# EPICS substitutions: template/mch_type1_ess.substitutions
#
# Type 1 : MCH
#          This is the standard ESS MCH for 9U/3U MTCA crate
#
#
# MCH (0)
# Manufacturer(12)         : Schroff GmbH
# Board Name(37)           : Schroff MicroTCA Backplane horizontal
# Manufacturer(12)         : Schroff GmbH
# Product Name(22)         : Schroff MicroTCA Shelf
# NAT-MCH (3)
# Manufacturer(21)         : N.A.T. GmbH - Germany
# Board Name(07)           : NAT-MCH
# Clock (60)
# Manufacturer(21)         : N.A.T. GmbH - Germany
# Product Name(16)         : NAT-MCH-CLK-PHYS
# HubMod1 (61)
# Manufacturer(21)         : N.A.T. GmbH - Germany
# Product Name(15)         : PCIe Hub Module

# show_fru
#  0   MCH       M4    NMCH-CM
#  3   mcmc1     M4    NAT-MCH-MCMC
# 60   Clock1    M4    MCH-Clock
# 61   HubMod1   M4    MCH-PCIe

# nat> show_sensorinfo 0
# Sensor Information for NMCH-CM
# ==================================================================
#   #   SDRType  Sensor Entity Inst  Value   State    Name
# ------------------------------------------------------------------
#   -   MDevLoc          0xc2  0x66                    NMCH-CM
#   0   Compact  0xf0    0xc2  0x66  0x10              HS 000 CM
# ------------------------------------------------------------------
# nat> show_sensorinfo 3
# Sensor Information for FRU 3 / MCMC1
# ==================================================================
#   #   SDRType  Sensor Entity Inst  Value   State    Name
# ------------------------------------------------------------------
#   -   MDevLoc          0xc2  0x61                    NAT-MCH-MCMC
#   1   Full     Temp    0xc2  0x61  36 C       ok     Temp CPU
#   2   Full     Temp    0xc2  0x61  32 C       ok     Temp I/O
#   3   Compact  0xf2    0xc2  0x61  0x01              HotSwap
#   4   Compact  0x2b    0xc2  0x61  0x00              Version Change
#   5   Full     Voltage 0xc2  0x61  1.20 V     ok     Base 1.2V
#   6   Full     Voltage 0xc2  0x61  1.51 V     ok     Base 1.5V
#   7   Full     Voltage 0xc2  0x61  1.81 V     ok     Base 1.8V
#   8   Full     Voltage 0xc2  0x61  2.45 V     ok     Base 2.5V
#   9   Full     Voltage 0xc2  0x61  3.360 V    ok     Base 3.3V
#  10   Full     Voltage 0xc2  0x61  12.30 V    ok     Base 12V
#  11   Full     Current 0xc2  0x61  1.51 A     ok     Base Current
#  12   Compact  0xf0    0xc2  0x61  0x10              HS 003 MCMC1
# ------------------------------------------------------------------
# nat> show_sensorinfo 60
# Sensor Information for FRU 60 / CLK1
# ==================================================================
#   #   SDRType  Sensor Entity Inst  Value   State    Name
# ------------------------------------------------------------------
#   -   MDevLoc          0xc2  0x63                    MCH-Clock
#   1   Full     Temp    0xc2  0x63  32 C       ok     Temp DC/DC
#   2   Full     Temp    0xc2  0x63  37 C       ok     Temp DC/DC max
#   3   Full     Temp    0xc2  0x63  42 C       ok     Temp Mux
#   4   Full     Temp    0xc2  0x63  46 C       ok     Temp Mux max
#   5   Full     Voltage 0xc2  0x63  3.328 V    ok     3.3V
#   6   Full     Voltage 0xc2  0x63  12.06 V    ok     12V
# ------------------------------------------------------------------
# nat> show_sensorinfo 61
# Sensor Information for FRU 61 / HUB1
# ==================================================================
#   #   SDRType  Sensor Entity Inst  Value   State    Name
# ------------------------------------------------------------------
#   -   MDevLoc          0xc2  0x64                    MCH-PCIe
#   1   Full     Temp    0xc2  0x64  33 C       ok     Temp DC/DC
#   2   Full     Temp    0xc2  0x64  38 C       ok     Temp DC/DC max
#   3   Full     Temp    0xc2  0x64  52 C       ok     Temp Switch
#   4   Full     Temp    0xc2  0x64  57 C       ok     Temp Switch max
#   5   Full     Temp    0xc2  0x64  34 C       ok     Temp PCB
#   6   Full     Temp    0xc2  0x64  30 C       ok     Temp PCB max
#   7   Full     Voltage 0xc2  0x64  0.90 V     ok     0.9V
#   8   Full     Voltage 0xc2  0x64  0.90 V     ok     0.9V analog
#   9   Full     Voltage 0xc2  0x64  1.80 V     ok     1.8V
#  10   Full     Voltage 0xc2  0x64  3.392 V    ok     3.3V
#  11   Full     Voltage 0xc2  0x64  12.30 V    ok     12V
# ------------------------------------------------------------------

global {dev=$(dev), unit=$(unit)}

file "fru_common_ess.template"
{
pattern { id,       fruid   }
        { MCHCM,    0       }
        { MCH,      3       }
        { CLK,      60      }
        { HUB,      61      }
}

file "sensor_ai_ess.template"
{
pattern { id,   fruid,  attr,       sensinst,   type,   prefix          }
        { MCH,  3,      CpuTemp,    1,          1,      $(id)$(unit)    }
        { MCH,  3,      IoTemp,     2,          1,      $(id)$(unit)    }
        { MCH,  3,      Base1d2V,   1,          2,      $(id)$(unit)    }
        { MCH,  3,      Base1d5V,   2,          2,      $(id)$(unit)    }
        { MCH,  3,      Base1d8V,   3,          2,      $(id)$(unit)    }
        { MCH,  3,      Base2d5V,   4,          2,      $(id)$(unit)    }
        { MCH,  3,      Base3d3V,   5,          2,      $(id)$(unit)    }
        { MCH,  3,      Base12V,    6,          2,      $(id)$(unit)    }
        { MCH,  3,      BaseI,      1,          3,      $(id)$(unit)    }
        { CLK,  60,     DcTemp,     1,          1,      $(id)$(unit)    }
        { CLK,  60,     DcMaxTemp,  2,          1,      $(id)$(unit)    }
        { CLK,  60,     MuxTemp,    3,          1,      $(id)$(unit)    }
        { CLK,  60,     MuxMaxTemp, 4,          1,      $(id)$(unit)    }
        { CLK,  60,     3d3V,       1,          2,      $(id)$(unit)    }
        { CLK,  60,     12V,        2,          2,      $(id)$(unit)    }
        { HUB,  61,     DcTemp,     1,          1,      $(id)$(unit)    }
        { HUB,  61,     DcMaxTemp,  2,          1,      $(id)$(unit)    }
        { HUB,  61,     SwTemp,     3,          1,      $(id)$(unit)    }
        { HUB,  61,     SwMaxTemp,  4,          1,      $(id)$(unit)    }
        { HUB,  61,     PcbTemp,    5,          1,      $(id)$(unit)    }
        { HUB,  61,     PcbMaxTemp, 6,          1,      $(id)$(unit)    }
        { HUB,  61,     d9V,        1,          2,      $(id)$(unit)    }
        { HUB,  61,     d9AnaV,     2,          2,      $(id)$(unit)    }
        { HUB,  61,     1d8V,       3,          2,      $(id)$(unit)    }
        { HUB,  61,     3d3V,       4,          2,      $(id)$(unit)    }
        { HUB,  61,     12V,        5,          2,      $(id)$(unit)    }
}
